RoboDK station: kr30 cnc_Test01.rdk

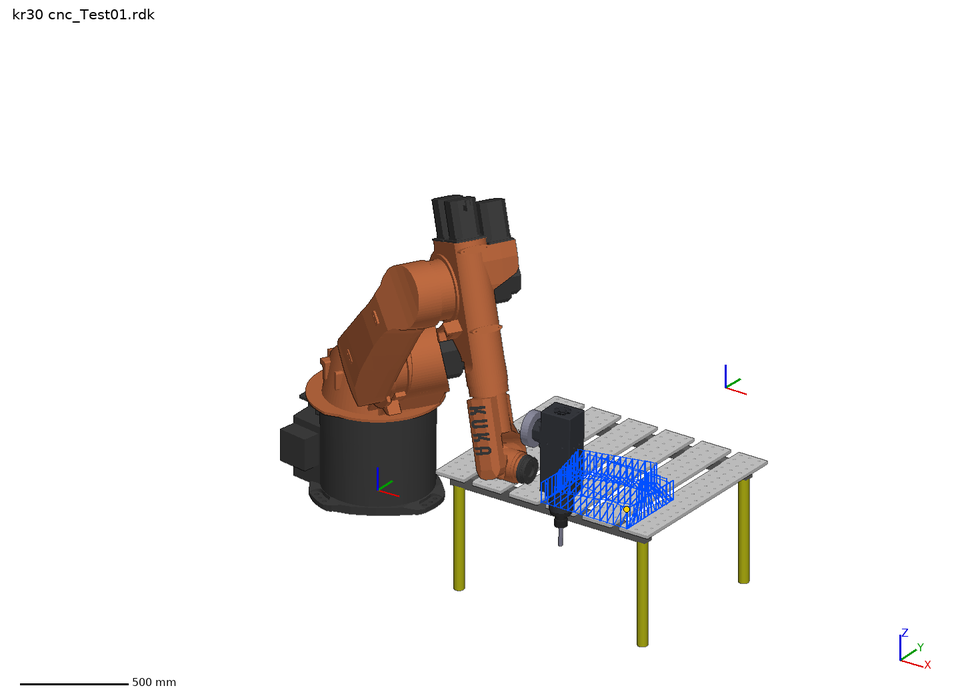
[picture v0: the station drawn from its stored meshes, robots at their saved joint values, targets as dots, program paths as lines]
Station kr30 cnc_Test01. Poses are relative to the parent item; angles as X-Y-Z fixed-axis rotations.
  - frame KUKA KR 30 HA Base at (0, 0, 0) mm
    - robot KUKA KR 30 HA: 6 axes, payload 30 kg, reach 2033 mm, repeatability 0.05 mm, weight 665 kg
        modified DH rows (alpha deg, a mm, theta deg, d mm): 0, 0, 0, 815; -90, 350, 0, 0; 0, 850, -90, 0; -90, 145, 0, 820; 90, 0, 0, 0; -90, 0, 180, 170
        joint limits [-185, -135, -120, -350, -119, -350] to [185, 35, 158, 350, 119, 350]; home [0, -90, 90, 0, 0, 0]; saved at [30.345, -48.669, 117.571, 35.552, -71.774, -11.781]
      - tool 1/2" End Mill TCP, TCP at (337.71, -2.2, 160.57) mm, size 692.9 x 170 x 256 mm
  - frame Milling Reference at (1256.02, 1000, 476.5) mm
    - object TABLE HEIGHT NOT YET SET at (0, -1000, 0) mm, size 1193.8 x 965.2 x 609.6 mm, geometry from welding_table.sld
    - object RhinoPart at (0, 0, 0) mm
  - machining project Machining Settings: rotZ(0) | rotX(0)*rotY(0) | rotZ(0) | onStart | onPathStart | onApproach | onPoint | onRetract | onFinish | Extruder(%1) | default | default | OutOnMov(%1) | OutOffMov(%1) | onPathFinish | M_RunCode(%1)
  - machining project RhinoPart Settings: rotZ(0) | rotX(0)*rotY(0) | roty(-90) | onStart | onPathStart | onApproach | onPoint | onRetract | onFinish | SetRPM(%1) | SetTool(%1) | Extruder(%1) | default | default | OutOnMov(%1) | OutOffMov(%1) | onPathFinish | M_RunCode(%1)
  - program RhinoPart (604 instructions, listed below)
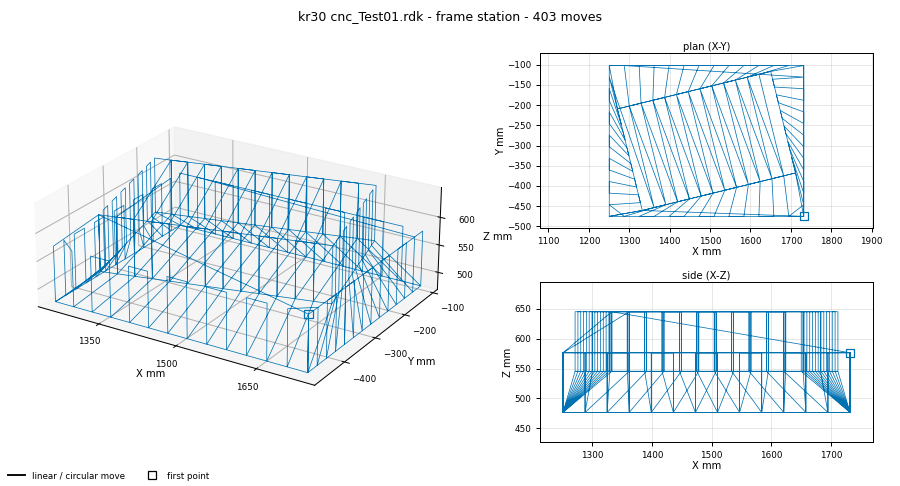
[picture p0: tool path of kr30 cnc_Test01.rdk in frame station, 403 of 403 moves have a stored position in this frame; points joined in program order, loops and branches not executed]

--- program RhinoPart (robot KUKA KR 30 HA) ---
  Set Ref.: Milling Reference
  Set Tool: 1/2" End Mill TCP
  Show 1/2" End Mill TCP
  Set speed (1000.0 mm/s)
  MoveJ 1 to (476.06, -1475.28, 100) mm, rotated rx 0 ry 90 rz 0 deg; joints [18.652, -58.205, 103.326, -154.528, 48.045, 162.335]
  MoveL 2 to (476.06, -1475.28, 100) mm, rotated rx 0 ry 90 rz 0 deg; joints [18.652, -58.205, 103.326, -154.528, 48.045, 162.335]
  MoveL 3 to (476.06, -1475.28, 0) mm, rotated rx 0 ry 90 rz 0 deg; joints [18.652, -54.047, 104.898, -156.478, 53.26, 165.406]
  MoveL 4 to (476.06, -1475.28, 0) mm, rotated rx 0 ry 90 rz 0 deg; joints [18.652, -54.047, 104.898, -156.478, 53.26, 165.406]
  Set speed (50.0 mm/s)
  MoveL 5 to (-5.57, -1475.28, 0) mm, rotated rx 0 ry 90 rz 0 deg; joints [27.216, -76.021, 140.928, -150.408, 67.844, 167.912]
  MoveL 6 to (-5.57, -1101.79, 0) mm, rotated rx 0 ry 90 rz 0 deg; joints [6.179, -81.84, 148.78, -173.289, 67.082, 177.377]
  MoveL 7 to (476.06, -1101.79, 0) mm, rotated rx 0 ry 90 rz 0 deg; joints [4.064, -57.785, 111.525, -174.964, 53.845, 177.024]
  MoveL 8 to (476.06, -1475.28, 0) mm, rotated rx 0 ry 90 rz 0 deg; joints [18.652, -54.047, 104.898, -156.478, 53.26, 165.406]
  Set speed (1000.0 mm/s)
  MoveL 9 to (476.06, -1475.28, 0) mm, rotated rx 0 ry 90 rz 0 deg; joints [18.652, -54.047, 104.898, -156.478, 53.26, 165.406]
  MoveL 10 to (476.06, -1475.28, 100) mm, rotated rx 0 ry 90 rz 0 deg; joints [18.652, -58.205, 103.326, -154.528, 48.045, 162.335]
  Set speed (1000.0 mm/s)
  MoveL 11 to (76.29, -1460.64, 168.91) mm, rotated rx 0 ry 90 rz 0 deg; joints [24.591, -82.592, 132.174, -148.989, 53.875, 160.486]
  MoveL 12 to (76.29, -1460.64, 68.91) mm, rotated rx 0 ry 90 rz 0 deg; joints [24.591, -77.019, 134.721, -151.568, 60.931, 165.262]
  MoveL 13 to (76.29, -1460.64, 68.91) mm, rotated rx 0 ry 90 rz 0 deg; joints [24.591, -77.019, 134.721, -151.568, 60.931, 165.262]
  Set speed (50.0 mm/s)
  MoveL 14 to (14.78, -1209.28, 68.91) mm, rotated rx 0 ry 90 rz 0 deg; joints [12.421, -85.064, 144.7, -165.681, 60.418, 172.818]
  MoveL 15 to (394.21, -1116.43, 68.91) mm, rotated rx 0 ry 90 rz 0 deg; joints [4.947, -65.156, 117.325, -173.745, 52.334, 176.169]
  MoveL 16 to (455.72, -1367.79, 68.91) mm, rotated rx 0 ry 90 rz 0 deg; joints [14.826, -59.674, 108.439, -160.608, 50.416, 167.358]
  MoveL 17 to (76.29, -1460.64, 68.91) mm, rotated rx 0 ry 90 rz 0 deg; joints [24.591, -77.019, 134.721, -151.568, 60.931, 165.262]
  Set speed (1000.0 mm/s)
  MoveL 18 to (76.29, -1460.64, 68.91) mm, rotated rx 0 ry 90 rz 0 deg; joints [24.591, -77.019, 134.721, -151.568, 60.931, 165.262]
  MoveL 19 to (76.29, -1460.64, 168.91) mm, rotated rx 0 ry 90 rz 0 deg; joints [24.591, -82.592, 132.174, -148.989, 53.875, 160.486]
  Set speed (1000.0 mm/s)
  MoveL 20 to (-5.57, -1475.28, 100) mm, rotated rx 0 ry 90 rz 0 deg; joints [27.216, -82.8, 138.885, -148.212, 60.252, 162.907]
  MoveL 21 to (-5.57, -1475.28, 0) mm, rotated rx 0 ry 90 rz 0 deg; joints [27.216, -76.021, 140.928, -150.408, 67.844, 167.912]
  MoveL 22 to (-5.57, -1475.28, 0) mm, rotated rx 0 ry 90 rz 0 deg; joints [27.216, -76.021, 140.928, -150.408, 67.844, 167.912]
  Set speed (50.0 mm/s)
  MoveL 23 to (76.29, -1460.64, 68.91) mm, rotated rx 0 ry 90 rz 0 deg; joints [24.591, -77.019, 134.721, -151.568, 60.931, 165.262]
  Set speed (1000.0 mm/s)
  MoveL 24 to (76.29, -1460.64, 68.91) mm, rotated rx 0 ry 90 rz 0 deg; joints [24.591, -77.019, 134.721, -151.568, 60.931, 165.262]
  MoveL 25 to (76.29, -1460.64, 168.91) mm, rotated rx 0 ry 90 rz 0 deg; joints [24.591, -82.592, 132.174, -148.989, 53.875, 160.486]
  Set speed (1000.0 mm/s)
  MoveL 26 to (455.72, -1367.79, 168.91) mm, rotated rx 0 ry 90 rz 0 deg; joints [14.826, -63.639, 106.295, -158.662, 44.688, 164.478]
  MoveL 27 to (455.72, -1367.79, 68.91) mm, rotated rx 0 ry 90 rz 0 deg; joints [14.826, -59.674, 108.439, -160.608, 50.416, 167.358]
  MoveL 28 to (455.72, -1367.79, 68.91) mm, rotated rx 0 ry 90 rz 0 deg; joints [14.826, -59.674, 108.439, -160.608, 50.416, 167.358]
  Set speed (50.0 mm/s)
  MoveL 29 to (476.06, -1475.28, 0) mm, rotated rx 0 ry 90 rz 0 deg; joints [18.652, -54.047, 104.898, -156.478, 53.26, 165.406]
  Set speed (1000.0 mm/s)
  MoveL 30 to (476.06, -1475.28, 0) mm, rotated rx 0 ry 90 rz 0 deg; joints [18.652, -54.047, 104.898, -156.478, 53.26, 165.406]
  MoveL 31 to (476.06, -1475.28, 100) mm, rotated rx 0 ry 90 rz 0 deg; joints [18.652, -58.205, 103.326, -154.528, 48.045, 162.335]
  Set speed (1000.0 mm/s)
  MoveL 32 to (476.06, -1101.79, 100) mm, rotated rx 0 ry 90 rz 0 deg; joints [4.064, -62.258, 109.929, -174.51, 47.803, 176.306]
  MoveL 33 to (476.06, -1101.79, 0) mm, rotated rx 0 ry 90 rz 0 deg; joints [4.064, -57.785, 111.525, -174.964, 53.845, 177.024]
  MoveL 34 to (476.06, -1101.79, 0) mm, rotated rx 0 ry 90 rz 0 deg; joints [4.064, -57.785, 111.525, -174.964, 53.845, 177.024]
  Set speed (50.0 mm/s)
  MoveL 35 to (394.21, -1116.43, 68.91) mm, rotated rx 0 ry 90 rz 0 deg; joints [4.947, -65.156, 117.325, -173.745, 52.334, 176.169]
  Set speed (1000.0 mm/s)
  MoveL 36 to (394.21, -1116.43, 68.91) mm, rotated rx 0 ry 90 rz 0 deg; joints [4.947, -65.156, 117.325, -173.745, 52.334, 176.169]
  MoveL 37 to (394.21, -1116.43, 168.91) mm, rotated rx 0 ry 90 rz 0 deg; joints [4.947, -69.559, 115.111, -173.086, 45.761, 175.165]
  Set speed (1000.0 mm/s)
  MoveL 38 to (14.78, -1209.28, 168.91) mm, rotated rx 0 ry 90 rz 0 deg; joints [12.421, -91.594, 141.782, -164.002, 51.297, 169.836]
  MoveL 39 to (14.78, -1209.28, 68.91) mm, rotated rx 0 ry 90 rz 0 deg; joints [12.421, -85.064, 144.7, -165.681, 60.418, 172.818]
  MoveL 40 to (14.78, -1209.28, 68.91) mm, rotated rx 0 ry 90 rz 0 deg; joints [12.421, -85.064, 144.7, -165.681, 60.418, 172.818]
  Set speed (50.0 mm/s)
  MoveL 41 to (-5.57, -1101.79, 0) mm, rotated rx 0 ry 90 rz 0 deg; joints [6.179, -81.84, 148.78, -173.289, 67.082, 177.377]
  Set speed (1000.0 mm/s)
  MoveL 42 to (-5.57, -1101.79, 0) mm, rotated rx 0 ry 90 rz 0 deg; joints [6.179, -81.84, 148.78, -173.289, 67.082, 177.377]
  MoveL 43 to (-5.57, -1101.79, 100) mm, rotated rx 0 ry 90 rz 0 deg; joints [6.179, -89.702, 146.455, -172.624, 56.97, 175.964]
  Set speed (1000.0 mm/s)
  MoveL 44 to (439.01, -1101.79, 100) mm, rotated rx 0 ry 90 rz 0 deg; joints [4.174, -64.255, 113.094, -174.463, 48.972, 176.359]
  MoveL 45 to (439.01, -1101.79, 0) mm, rotated rx 0 ry 90 rz 0 deg; joints [4.174, -59.613, 114.709, -174.914, 55.202, 177.093]
  MoveL 46 to (439.01, -1101.79, 0) mm, rotated rx 0 ry 90 rz 0 deg; joints [4.174, -59.613, 114.709, -174.914, 55.202, 177.093]
  Set speed (50.0 mm/s)
  MoveL 47 to (365.02, -1123.57, 68.91) mm, rotated rx 0 ry 90 rz 0 deg; joints [5.373, -66.644, 119.654, -173.284, 53.2, 175.965]
  Set speed (1000.0 mm/s)
  MoveL 48 to (365.02, -1123.57, 68.91) mm, rotated rx 0 ry 90 rz 0 deg; joints [5.373, -66.644, 119.654, -173.284, 53.2, 175.965]
  MoveL 49 to (365.02, -1123.57, 168.91) mm, rotated rx 0 ry 90 rz 0 deg; joints [5.373, -71.176, 117.413, -172.58, 46.477, 174.875]
  Set speed (1000.0 mm/s)
  MoveL 50 to (335.84, -1130.72, 168.91) mm, rotated rx 0 ry 90 rz 0 deg; joints [5.818, -72.795, 119.668, -172.052, 47.149, 174.576]
  MoveL 51 to (335.84, -1130.72, 68.91) mm, rotated rx 0 ry 90 rz 0 deg; joints [5.818, -68.13, 121.942, -172.805, 54.028, 175.759]
  MoveL 52 to (335.84, -1130.72, 68.91) mm, rotated rx 0 ry 90 rz 0 deg; joints [5.818, -68.13, 121.942, -172.805, 54.028, 175.759]
  Set speed (50.0 mm/s)
  MoveL 53 to (401.97, -1101.79, 0) mm, rotated rx 0 ry 90 rz 0 deg; joints [4.29, -61.424, 117.823, -174.853, 56.506, 177.154]
  Set speed (1000.0 mm/s)
  MoveL 54 to (401.97, -1101.79, 0) mm, rotated rx 0 ry 90 rz 0 deg; joints [4.29, -61.424, 117.823, -174.853, 56.506, 177.154]
  MoveL 55 to (401.97, -1101.79, 100) mm, rotated rx 0 ry 90 rz 0 deg; joints [4.29, -66.245, 116.184, -174.402, 50.074, 176.4]
  Set speed (1000.0 mm/s)
  MoveL 56 to (364.92, -1101.79, 100) mm, rotated rx 0 ry 90 rz 0 deg; joints [4.413, -68.234, 119.205, -174.326, 51.109, 176.431]
  MoveL 57 to (364.92, -1101.79, 0) mm, rotated rx 0 ry 90 rz 0 deg; joints [4.413, -63.224, 120.874, -174.78, 57.758, 177.21]
  MoveL 58 to (364.92, -1101.79, 0) mm, rotated rx 0 ry 90 rz 0 deg; joints [4.413, -63.224, 120.874, -174.78, 57.758, 177.21]
  Set speed (50.0 mm/s)
  MoveL 59 to (306.65, -1137.86, 68.91) mm, rotated rx 0 ry 90 rz 0 deg; joints [6.283, -69.615, 124.19, -172.305, 54.819, 175.548]
  Set speed (1000.0 mm/s)
  MoveL 60 to (306.65, -1137.86, 68.91) mm, rotated rx 0 ry 90 rz 0 deg; joints [6.283, -69.615, 124.19, -172.305, 54.819, 175.548]
  MoveL 61 to (306.65, -1137.86, 168.91) mm, rotated rx 0 ry 90 rz 0 deg; joints [6.283, -74.42, 121.88, -171.501, 47.775, 174.265]
  Set speed (1000.0 mm/s)
  MoveL 62 to (277.46, -1145, 168.91) mm, rotated rx 0 ry 90 rz 0 deg; joints [6.77, -76.052, 124.049, -170.924, 48.355, 173.94]
  MoveL 63 to (277.46, -1145, 68.91) mm, rotated rx 0 ry 90 rz 0 deg; joints [6.77, -71.103, 126.399, -171.783, 55.572, 175.333]
  MoveL 64 to (277.46, -1145, 68.91) mm, rotated rx 0 ry 90 rz 0 deg; joints [6.77, -71.103, 126.399, -171.783, 55.572, 175.333]
  Set speed (50.0 mm/s)
  MoveL 65 to (327.87, -1101.79, 0) mm, rotated rx 0 ry 90 rz 0 deg; joints [4.543, -65.017, 123.867, -174.696, 58.958, 177.259]
  Set speed (1000.0 mm/s)
  MoveL 66 to (327.87, -1101.79, 0) mm, rotated rx 0 ry 90 rz 0 deg; joints [4.543, -65.017, 123.867, -174.696, 58.958, 177.259]
  MoveL 67 to (327.87, -1101.79, 100) mm, rotated rx 0 ry 90 rz 0 deg; joints [4.543, -70.229, 122.163, -174.237, 52.075, 176.45]
  Set speed (1000.0 mm/s)
  MoveL 68 to (290.82, -1101.79, 100) mm, rotated rx 0 ry 90 rz 0 deg; joints [4.681, -72.237, 125.063, -174.133, 52.971, 176.459]
  MoveL 69 to (290.82, -1101.79, 0) mm, rotated rx 0 ry 90 rz 0 deg; joints [4.681, -66.809, 126.806, -174.599, 60.107, 177.302]
  MoveL 70 to (290.82, -1101.79, 0) mm, rotated rx 0 ry 90 rz 0 deg; joints [4.681, -66.809, 126.806, -174.599, 60.107, 177.302]
  Set speed (50.0 mm/s)
  MoveL 71 to (248.28, -1152.14, 68.91) mm, rotated rx 0 ry 90 rz 0 deg; joints [7.28, -72.596, 128.57, -171.237, 56.285, 175.11]
  Set speed (1000.0 mm/s)
  MoveL 72 to (248.28, -1152.14, 68.91) mm, rotated rx 0 ry 90 rz 0 deg; joints [7.28, -72.596, 128.57, -171.237, 56.285, 175.11]
  MoveL 73 to (248.28, -1152.14, 168.91) mm, rotated rx 0 ry 90 rz 0 deg; joints [7.28, -77.695, 126.177, -170.317, 48.889, 173.599]
  Set speed (1000.0 mm/s)
  MoveL 74 to (219.09, -1159.28, 168.91) mm, rotated rx 0 ry 90 rz 0 deg; joints [7.815, -79.352, 128.264, -169.68, 49.375, 173.238]
  MoveL 75 to (219.09, -1159.28, 68.91) mm, rotated rx 0 ry 90 rz 0 deg; joints [7.815, -74.097, 130.706, -170.665, 56.959, 174.878]
  MoveL 76 to (219.09, -1159.28, 68.91) mm, rotated rx 0 ry 90 rz 0 deg; joints [7.815, -74.097, 130.706, -170.665, 56.959, 174.878]
  Set speed (50.0 mm/s)
  MoveL 77 to (253.77, -1101.79, 0) mm, rotated rx 0 ry 90 rz 0 deg; joints [4.827, -68.606, 129.696, -174.489, 61.202, 177.339]
  Set speed (1000.0 mm/s)
  MoveL 78 to (253.77, -1101.79, 0) mm, rotated rx 0 ry 90 rz 0 deg; joints [4.827, -68.606, 129.696, -174.489, 61.202, 177.339]
  MoveL 79 to (253.77, -1101.79, 100) mm, rotated rx 0 ry 90 rz 0 deg; joints [4.827, -74.263, 127.907, -174.014, 53.793, 176.455]
  Set speed (1000.0 mm/s)
  MoveL 80 to (216.72, -1101.79, 100) mm, rotated rx 0 ry 90 rz 0 deg; joints [4.983, -76.315, 130.699, -173.878, 54.538, 176.439]
  MoveL 81 to (216.72, -1101.79, 0) mm, rotated rx 0 ry 90 rz 0 deg; joints [4.983, -70.411, 132.54, -174.367, 62.243, 177.37]
  MoveL 82 to (216.72, -1101.79, 0) mm, rotated rx 0 ry 90 rz 0 deg; joints [4.983, -70.411, 132.54, -174.367, 62.243, 177.37]
  Set speed (50.0 mm/s)
  MoveL 83 to (189.9, -1166.42, 68.91) mm, rotated rx 0 ry 90 rz 0 deg; joints [8.376, -75.608, 132.806, -170.064, 57.591, 174.637]
  Set speed (1000.0 mm/s)
  MoveL 84 to (189.9, -1166.42, 68.91) mm, rotated rx 0 ry 90 rz 0 deg; joints [8.376, -75.608, 132.806, -170.064, 57.591, 174.637]
  MoveL 85 to (189.9, -1166.42, 168.91) mm, rotated rx 0 ry 90 rz 0 deg; joints [8.376, -81.025, 130.312, -169.007, 49.811, 172.855]
  Set speed (1000.0 mm/s)
  MoveL 86 to (160.71, -1173.57, 168.91) mm, rotated rx 0 ry 90 rz 0 deg; joints [8.966, -82.718, 132.321, -168.296, 50.196, 172.445]
  MoveL 87 to (160.71, -1173.57, 68.91) mm, rotated rx 0 ry 90 rz 0 deg; joints [8.966, -77.132, 134.873, -169.432, 58.181, 174.382]
  MoveL 88 to (160.71, -1173.57, 68.91) mm, rotated rx 0 ry 90 rz 0 deg; joints [8.966, -77.132, 134.873, -169.432, 58.181, 174.382]
  Set speed (50.0 mm/s)
  MoveL 89 to (179.68, -1101.79, 0) mm, rotated rx 0 ry 90 rz 0 deg; joints [5.149, -72.232, 135.341, -174.23, 63.226, 177.394]
  Set speed (1000.0 mm/s)
  MoveL 90 to (179.68, -1101.79, 0) mm, rotated rx 0 ry 90 rz 0 deg; joints [5.149, -72.232, 135.341, -174.23, 63.226, 177.394]
  MoveL 91 to (179.68, -1101.79, 100) mm, rotated rx 0 ry 90 rz 0 deg; joints [5.149, -78.402, 133.441, -173.725, 55.2, 176.409]
  Set speed (1000.0 mm/s)
  MoveL 92 to (142.63, -1101.79, 100) mm, rotated rx 0 ry 90 rz 0 deg; joints [5.327, -80.532, 136.135, -173.553, 55.773, 176.363]
  MoveL 93 to (142.63, -1101.79, 0) mm, rotated rx 0 ry 90 rz 0 deg; joints [5.327, -74.075, 138.101, -174.079, 64.146, 177.41]
  MoveL 94 to (142.63, -1101.79, 0) mm, rotated rx 0 ry 90 rz 0 deg; joints [5.327, -74.075, 138.101, -174.079, 64.146, 177.41]
  Set speed (50.0 mm/s)
  MoveL 95 to (131.53, -1180.71, 68.91) mm, rotated rx 0 ry 90 rz 0 deg; joints [9.586, -78.673, 136.905, -168.765, 58.727, 174.112]
  Set speed (1000.0 mm/s)
  MoveL 96 to (131.53, -1180.71, 68.91) mm, rotated rx 0 ry 90 rz 0 deg; joints [9.586, -78.673, 136.905, -168.765, 58.727, 174.112]
  MoveL 97 to (131.53, -1180.71, 168.91) mm, rotated rx 0 ry 90 rz 0 deg; joints [9.586, -84.433, 134.291, -167.542, 50.529, 172.006]
  Set speed (1000.0 mm/s)
  MoveL 98 to (102.34, -1187.85, 168.91) mm, rotated rx 0 ry 90 rz 0 deg; joints [10.239, -86.175, 136.223, -166.741, 50.808, 171.531]
  MoveL 99 to (102.34, -1187.85, 68.91) mm, rotated rx 0 ry 90 rz 0 deg; joints [10.239, -80.232, 138.904, -168.06, 59.225, 173.825]
  MoveL 100 to (102.34, -1187.85, 68.91) mm, rotated rx 0 ry 90 rz 0 deg; joints [10.239, -80.232, 138.904, -168.06, 59.225, 173.825]
  Set speed (50.0 mm/s)
  MoveL 101 to (105.58, -1101.79, 0) mm, rotated rx 0 ry 90 rz 0 deg; joints [5.517, -75.948, 140.824, -173.91, 65, 177.418]
  Set speed (1000.0 mm/s)
  MoveL 102 to (105.58, -1101.79, 0) mm, rotated rx 0 ry 90 rz 0 deg; joints [5.517, -75.948, 140.824, -173.91, 65, 177.418]
  MoveL 103 to (105.58, -1101.79, 100) mm, rotated rx 0 ry 90 rz 0 deg; joints [5.517, -82.714, 138.783, -173.36, 56.248, 176.299]
  Set speed (1000.0 mm/s)
  MoveL 104 to (68.53, -1101.79, 100) mm, rotated rx 0 ry 90 rz 0 deg; joints [5.721, -84.961, 141.386, -173.143, 56.614, 176.214]
  MoveL 105 to (68.53, -1101.79, 0) mm, rotated rx 0 ry 90 rz 0 deg; joints [5.721, -77.859, 143.51, -173.724, 65.78, 177.417]
  MoveL 106 to (68.53, -1101.79, 0) mm, rotated rx 0 ry 90 rz 0 deg; joints [5.721, -77.859, 143.51, -173.724, 65.78, 177.417]
  Set speed (50.0 mm/s)
  MoveL 107 to (73.15, -1194.99, 68.91) mm, rotated rx 0 ry 90 rz 0 deg; joints [10.927, -81.815, 140.87, -167.314, 59.675, 173.516]
  Set speed (1000.0 mm/s)
  MoveL 108 to (73.15, -1194.99, 68.91) mm, rotated rx 0 ry 90 rz 0 deg; joints [10.927, -81.815, 140.87, -167.314, 59.675, 173.516]
  MoveL 109 to (73.15, -1194.99, 168.91) mm, rotated rx 0 ry 90 rz 0 deg; joints [10.927, -87.947, 138.116, -165.888, 51.03, 171.015]
  Set speed (1000.0 mm/s)
  MoveL 110 to (43.97, -1202.13, 168.91) mm, rotated rx 0 ry 90 rz 0 deg; joints [11.653, -89.752, 139.969, -164.977, 51.194, 170.453]
  MoveL 111 to (43.97, -1202.13, 68.91) mm, rotated rx 0 ry 90 rz 0 deg; joints [11.653, -83.424, 142.801, -166.522, 60.074, 173.182]
  MoveL 112 to (43.97, -1202.13, 68.91) mm, rotated rx 0 ry 90 rz 0 deg; joints [11.653, -83.424, 142.801, -166.522, 60.074, 173.182]
  Set speed (50.0 mm/s)
  MoveL 113 to (31.48, -1101.79, 0) mm, rotated rx 0 ry 90 rz 0 deg; joints [5.941, -79.819, 146.162, -173.518, 66.477, 177.404]
  Set speed (1000.0 mm/s)
  MoveL 114 to (31.48, -1101.79, 0) mm, rotated rx 0 ry 90 rz 0 deg; joints [5.941, -79.819, 146.162, -173.518, 66.477, 177.404]
  MoveL 115 to (31.48, -1101.79, 100) mm, rotated rx 0 ry 90 rz 0 deg; joints [5.941, -87.285, 143.943, -172.899, 56.86, 176.104]
  Set speed (1000.0 mm/s)
  MoveL 116 to (476.06, -1130.52, 100) mm, rotated rx 0 ry 90 rz 0 deg; joints [5.231, -62.132, 109.727, -172.932, 47.813, 175.24]
  MoveL 117 to (476.06, -1130.52, 0) mm, rotated rx 0 ry 90 rz 0 deg; joints [5.231, -57.67, 111.322, -173.515, 53.828, 176.162]
  MoveL 118 to (476.06, -1130.52, 0) mm, rotated rx 0 ry 90 rz 0 deg; joints [5.231, -57.67, 111.322, -173.515, 53.828, 176.162]
  Set speed (50.0 mm/s)
  MoveL 119 to (398.94, -1135.77, 68.91) mm, rotated rx 0 ry 90 rz 0 deg; joints [5.759, -64.815, 116.785, -172.704, 52.196, 175.513]
  Set speed (1000.0 mm/s)
  MoveL 120 to (398.94, -1135.77, 68.91) mm, rotated rx 0 ry 90 rz 0 deg; joints [5.759, -64.815, 116.785, -172.704, 52.196, 175.513]
  MoveL 121 to (398.94, -1135.77, 168.91) mm, rotated rx 0 ry 90 rz 0 deg; joints [5.759, -69.188, 114.577, -171.937, 45.673, 174.347]
  Set speed (1000.0 mm/s)
  MoveL 122 to (403.67, -1155.1, 168.91) mm, rotated rx 0 ry 90 rz 0 deg; joints [6.563, -68.804, 114.02, -170.793, 45.588, 173.529]
  MoveL 123 to (403.67, -1155.1, 68.91) mm, rotated rx 0 ry 90 rz 0 deg; joints [6.563, -64.46, 116.222, -171.667, 52.057, 174.854]
  MoveL 124 to (403.67, -1155.1, 68.91) mm, rotated rx 0 ry 90 rz 0 deg; joints [6.563, -64.46, 116.222, -171.667, 52.057, 174.854]
  Set speed (50.0 mm/s)
  MoveL 125 to (476.06, -1159.25, 0) mm, rotated rx 0 ry 90 rz 0 deg; joints [6.394, -57.525, 111.068, -172.069, 53.806, 175.297]
  Set speed (1000.0 mm/s)
  MoveL 126 to (476.06, -1159.25, 0) mm, rotated rx 0 ry 90 rz 0 deg; joints [6.394, -57.525, 111.068, -172.069, 53.806, 175.297]
  MoveL 127 to (476.06, -1159.25, 100) mm, rotated rx 0 ry 90 rz 0 deg; joints [6.394, -61.974, 109.474, -171.358, 47.826, 174.174]
  Set speed (1000.0 mm/s)
  MoveL 128 to (476.06, -1187.98, 100) mm, rotated rx 0 ry 90 rz 0 deg; joints [7.551, -61.785, 109.171, -169.789, 47.841, 173.107]
  MoveL 129 to (476.06, -1187.98, 0) mm, rotated rx 0 ry 90 rz 0 deg; joints [7.551, -57.351, 110.763, -170.626, 53.78, 174.428]
  MoveL 130 to (476.06, -1187.98, 0) mm, rotated rx 0 ry 90 rz 0 deg; joints [7.551, -57.351, 110.763, -170.626, 53.78, 174.428]
  Set speed (50.0 mm/s)
  MoveL 131 to (408.4, -1174.44, 68.91) mm, rotated rx 0 ry 90 rz 0 deg; joints [7.358, -64.091, 115.634, -170.636, 51.917, 174.192]
  Set speed (1000.0 mm/s)
  MoveL 132 to (408.4, -1174.44, 68.91) mm, rotated rx 0 ry 90 rz 0 deg; joints [7.358, -64.091, 115.634, -170.636, 51.917, 174.192]
  MoveL 133 to (408.4, -1174.44, 168.91) mm, rotated rx 0 ry 90 rz 0 deg; joints [7.358, -68.404, 113.438, -169.657, 45.504, 172.711]
  Set speed (1000.0 mm/s)
  MoveL 134 to (413.14, -1193.77, 168.91) mm, rotated rx 0 ry 90 rz 0 deg; joints [8.145, -67.99, 112.833, -168.527, 45.421, 171.893]
  MoveL 135 to (413.14, -1193.77, 68.91) mm, rotated rx 0 ry 90 rz 0 deg; joints [8.145, -63.709, 115.023, -169.61, 51.775, 173.528]
  MoveL 136 to (413.14, -1193.77, 68.91) mm, rotated rx 0 ry 90 rz 0 deg; joints [8.145, -63.709, 115.023, -169.61, 51.775, 173.528]
  Set speed (50.0 mm/s)
  MoveL 137 to (476.06, -1216.71, 0) mm, rotated rx 0 ry 90 rz 0 deg; joints [8.702, -57.148, 110.406, -169.187, 53.749, 173.556]
  Set speed (1000.0 mm/s)
  MoveL 138 to (476.06, -1216.71, 0) mm, rotated rx 0 ry 90 rz 0 deg; joints [8.702, -57.148, 110.406, -169.187, 53.749, 173.556]
  MoveL 139 to (476.06, -1216.71, 100) mm, rotated rx 0 ry 90 rz 0 deg; joints [8.702, -61.564, 108.816, -168.227, 47.858, 172.039]
  Set speed (1000.0 mm/s)
  MoveL 140 to (476.06, -1245.44, 100) mm, rotated rx 0 ry 90 rz 0 deg; joints [9.846, -61.313, 108.41, -166.671, 47.877, 170.97]
  MoveL 141 to (476.06, -1245.44, 0) mm, rotated rx 0 ry 90 rz 0 deg; joints [9.846, -56.917, 109.999, -167.752, 53.713, 172.679]
  MoveL 142 to (476.06, -1245.44, 0) mm, rotated rx 0 ry 90 rz 0 deg; joints [9.846, -56.917, 109.999, -167.752, 53.713, 172.679]
  Set speed (50.0 mm/s)
  MoveL 143 to (417.87, -1213.11, 68.91) mm, rotated rx 0 ry 90 rz 0 deg; joints [8.923, -63.313, 114.388, -168.59, 51.633, 172.86]
  Set speed (1000.0 mm/s)
  MoveL 144 to (417.87, -1213.11, 68.91) mm, rotated rx 0 ry 90 rz 0 deg; joints [8.923, -63.313, 114.388, -168.59, 51.633, 172.86]
  MoveL 145 to (417.87, -1213.11, 168.91) mm, rotated rx 0 ry 90 rz 0 deg; joints [8.923, -67.561, 112.203, -167.405, 45.34, 171.074]
  Set speed (1000.0 mm/s)
  MoveL 146 to (422.6, -1232.44, 168.91) mm, rotated rx 0 ry 90 rz 0 deg; joints [9.693, -67.119, 111.55, -166.289, 45.259, 170.255]
  MoveL 147 to (422.6, -1232.44, 68.91) mm, rotated rx 0 ry 90 rz 0 deg; joints [9.693, -62.904, 113.728, -167.575, 51.488, 172.188]
  MoveL 148 to (422.6, -1232.44, 68.91) mm, rotated rx 0 ry 90 rz 0 deg; joints [9.693, -62.904, 113.728, -167.575, 51.488, 172.188]
  Set speed (50.0 mm/s)
  MoveL 149 to (476.06, -1274.17, 0) mm, rotated rx 0 ry 90 rz 0 deg; joints [10.982, -56.657, 109.54, -166.322, 53.673, 171.797]
  Set speed (1000.0 mm/s)
  MoveL 150 to (476.06, -1274.17, 0) mm, rotated rx 0 ry 90 rz 0 deg; joints [10.982, -56.657, 109.54, -166.322, 53.673, 171.797]
  MoveL 151 to (476.06, -1274.17, 100) mm, rotated rx 0 ry 90 rz 0 deg; joints [10.982, -61.03, 107.954, -165.122, 47.897, 169.9]
  Set speed (1000.0 mm/s)
  MoveL 152 to (476.06, -1302.9, 100) mm, rotated rx 0 ry 90 rz 0 deg; joints [12.109, -60.717, 107.446, -163.581, 47.918, 168.829]
  MoveL 153 to (476.06, -1302.9, 0) mm, rotated rx 0 ry 90 rz 0 deg; joints [12.109, -56.368, 109.03, -164.898, 53.628, 170.908]
  MoveL 154 to (476.06, -1302.9, 0) mm, rotated rx 0 ry 90 rz 0 deg; joints [12.109, -56.368, 109.03, -164.898, 53.628, 170.908]
  Set speed (50.0 mm/s)
  MoveL 155 to (427.33, -1251.78, 68.91) mm, rotated rx 0 ry 90 rz 0 deg; joints [10.453, -62.481, 113.045, -166.565, 51.342, 171.513]
  Set speed (1000.0 mm/s)
  MoveL 156 to (427.33, -1251.78, 68.91) mm, rotated rx 0 ry 90 rz 0 deg; joints [10.453, -62.481, 113.045, -166.565, 51.342, 171.513]
  MoveL 157 to (427.33, -1251.78, 168.91) mm, rotated rx 0 ry 90 rz 0 deg; joints [10.453, -66.663, 110.872, -165.18, 45.178, 169.435]
  Set speed (1000.0 mm/s)
  MoveL 158 to (432.06, -1271.11, 168.91) mm, rotated rx 0 ry 90 rz 0 deg; joints [11.205, -66.192, 110.17, -164.077, 45.098, 168.614]
  MoveL 159 to (432.06, -1271.11, 68.91) mm, rotated rx 0 ry 90 rz 0 deg; joints [11.205, -62.045, 112.337, -165.56, 51.193, 170.833]
  MoveL 160 to (432.06, -1271.11, 68.91) mm, rotated rx 0 ry 90 rz 0 deg; joints [11.205, -62.045, 112.337, -165.56, 51.193, 170.833]
  Set speed (50.0 mm/s)
  MoveL 161 to (476.06, -1331.63, 0) mm, rotated rx 0 ry 90 rz 0 deg; joints [13.228, -56.052, 108.47, -163.479, 53.579, 170.013]
  Set speed (1000.0 mm/s)
  MoveL 162 to (476.06, -1331.63, 0) mm, rotated rx 0 ry 90 rz 0 deg; joints [13.228, -56.052, 108.47, -163.479, 53.579, 170.013]
  MoveL 163 to (476.06, -1331.63, 100) mm, rotated rx 0 ry 90 rz 0 deg; joints [13.228, -60.373, 106.888, -162.049, 47.939, 167.755]
  Set speed (1000.0 mm/s)
  MoveL 164 to (476.06, -1360.36, 100) mm, rotated rx 0 ry 90 rz 0 deg; joints [14.335, -59.999, 106.278, -160.526, 47.961, 166.679]
  MoveL 165 to (476.06, -1360.36, 0) mm, rotated rx 0 ry 90 rz 0 deg; joints [14.335, -55.707, 107.858, -162.067, 53.525, 169.11]
  MoveL 166 to (476.06, -1360.36, 0) mm, rotated rx 0 ry 90 rz 0 deg; joints [14.335, -55.707, 107.858, -162.067, 53.525, 169.11]
  Set speed (50.0 mm/s)
  MoveL 167 to (436.79, -1290.45, 68.91) mm, rotated rx 0 ry 90 rz 0 deg; joints [11.948, -61.597, 111.606, -164.56, 51.043, 170.149]
  Set speed (1000.0 mm/s)
  MoveL 168 to (436.79, -1290.45, 68.91) mm, rotated rx 0 ry 90 rz 0 deg; joints [11.948, -61.597, 111.606, -164.56, 51.043, 170.149]
  MoveL 169 to (436.79, -1290.45, 168.91) mm, rotated rx 0 ry 90 rz 0 deg; joints [11.948, -65.709, 109.444, -162.982, 45.018, 167.791]
  Set speed (1000.0 mm/s)
  MoveL 170 to (441.52, -1309.79, 168.91) mm, rotated rx 0 ry 90 rz 0 deg; joints [12.681, -65.211, 108.693, -161.893, 44.937, 166.967]
  MoveL 171 to (441.52, -1309.79, 68.91) mm, rotated rx 0 ry 90 rz 0 deg; joints [12.681, -61.135, 110.851, -163.566, 50.89, 169.459]
  MoveL 172 to (441.52, -1309.79, 68.91) mm, rotated rx 0 ry 90 rz 0 deg; joints [12.681, -61.135, 110.851, -163.566, 50.89, 169.459]
  Set speed (50.0 mm/s)
  MoveL 173 to (476.06, -1389.09, 0) mm, rotated rx 0 ry 90 rz 0 deg; joints [15.432, -55.334, 107.195, -160.66, 53.466, 168.198]
  Set speed (1000.0 mm/s)
  MoveL 174 to (476.06, -1389.09, 0) mm, rotated rx 0 ry 90 rz 0 deg; joints [15.432, -55.334, 107.195, -160.66, 53.466, 168.198]
  MoveL 175 to (476.06, -1389.09, 100) mm, rotated rx 0 ry 90 rz 0 deg; joints [15.432, -59.595, 105.617, -159.012, 47.983, 165.599]
  Set speed (1000.0 mm/s)
  MoveL 176 to (476.06, -1417.82, 100) mm, rotated rx 0 ry 90 rz 0 deg; joints [16.518, -59.161, 104.905, -157.508, 48.005, 164.516]
  MoveL 177 to (476.06, -1417.82, 0) mm, rotated rx 0 ry 90 rz 0 deg; joints [16.518, -54.933, 106.481, -159.259, 53.402, 167.278]
  MoveL 178 to (476.06, -1417.82, 0) mm, rotated rx 0 ry 90 rz 0 deg; joints [16.518, -54.933, 106.481, -159.259, 53.402, 167.278]
  Set speed (50.0 mm/s)
  MoveL 179 to (446.25, -1329.12, 68.91) mm, rotated rx 0 ry 90 rz 0 deg; joints [13.405, -60.661, 110.071, -162.575, 50.734, 168.765]
  Set speed (1000.0 mm/s)
  MoveL 180 to (446.25, -1329.12, 68.91) mm, rotated rx 0 ry 90 rz 0 deg; joints [13.405, -60.661, 110.071, -162.575, 50.734, 168.765]
  MoveL 181 to (446.25, -1329.12, 168.91) mm, rotated rx 0 ry 90 rz 0 deg; joints [13.405, -64.7, 107.919, -160.81, 44.855, 166.14]
  Set speed (1000.0 mm/s)
  MoveL 182 to (450.99, -1348.46, 168.91) mm, rotated rx 0 ry 90 rz 0 deg; joints [14.12, -64.176, 107.119, -159.733, 44.772, 165.311]
  MoveL 183 to (450.99, -1348.46, 68.91) mm, rotated rx 0 ry 90 rz 0 deg; joints [14.12, -60.174, 109.267, -161.59, 50.577, 168.065]
  MoveL 184 to (450.99, -1348.46, 68.91) mm, rotated rx 0 ry 90 rz 0 deg; joints [14.12, -60.174, 109.267, -161.59, 50.577, 168.065]
  Set speed (50.0 mm/s)
  MoveL 185 to (476.06, -1446.55, 0) mm, rotated rx 0 ry 90 rz 0 deg; joints [17.591, -54.504, 105.715, -157.865, 53.333, 166.347]
  Set speed (1000.0 mm/s)
  MoveL 186 to (476.06, -1446.55, 0) mm, rotated rx 0 ry 90 rz 0 deg; joints [17.591, -54.504, 105.715, -157.865, 53.333, 166.347]
  MoveL 187 to (476.06, -1446.55, 100) mm, rotated rx 0 ry 90 rz 0 deg; joints [17.591, -58.698, 104.141, -156.013, 48.025, 163.428]
  Set speed (1000.0 mm/s)
  MoveL 188 to (439.01, -1475.28, 100) mm, rotated rx 0 ry 90 rz 0 deg; joints [19.122, -60.131, 106.492, -154.402, 49.306, 162.653]
  MoveL 189 to (439.01, -1475.28, 0) mm, rotated rx 0 ry 90 rz 0 deg; joints [19.122, -55.828, 108.073, -156.321, 54.655, 165.765]
  MoveL 190 to (439.01, -1475.28, 0) mm, rotated rx 0 ry 90 rz 0 deg; joints [19.122, -55.828, 108.073, -156.321, 54.655, 165.765]
  Set speed (50.0 mm/s)
  MoveL 191 to (426.53, -1374.93, 68.91) mm, rotated rx 0 ry 90 rz 0 deg; joints [15.413, -61.068, 110.741, -160.118, 51.4, 167.286]
  Set speed (1000.0 mm/s)
  MoveL 192 to (426.53, -1374.93, 68.91) mm, rotated rx 0 ry 90 rz 0 deg; joints [15.413, -61.068, 110.741, -160.118, 51.4, 167.286]
  MoveL 193 to (426.53, -1374.93, 168.91) mm, rotated rx 0 ry 90 rz 0 deg; joints [15.413, -65.139, 108.584, -158.153, 45.579, 164.325]
  Set speed (1000.0 mm/s)
  MoveL 194 to (397.34, -1382.08, 168.91) mm, rotated rx 0 ry 90 rz 0 deg; joints [16.023, -66.626, 110.817, -157.609, 46.436, 164.149]
  MoveL 195 to (397.34, -1382.08, 68.91) mm, rotated rx 0 ry 90 rz 0 deg; joints [16.023, -62.447, 112.99, -159.597, 52.351, 167.2]
  MoveL 196 to (397.34, -1382.08, 68.91) mm, rotated rx 0 ry 90 rz 0 deg; joints [16.023, -62.447, 112.99, -159.597, 52.351, 167.2]
  Set speed (50.0 mm/s)
  MoveL 197 to (401.97, -1475.28, 0) mm, rotated rx 0 ry 90 rz 0 deg; joints [19.616, -57.579, 111.163, -156.113, 56, 166.09]
  Set speed (1000.0 mm/s)
  MoveL 198 to (401.97, -1475.28, 0) mm, rotated rx 0 ry 90 rz 0 deg; joints [19.616, -57.579, 111.163, -156.113, 56, 166.09]
  MoveL 199 to (401.97, -1475.28, 100) mm, rotated rx 0 ry 90 rz 0 deg; joints [19.616, -62.033, 109.569, -154.214, 50.51, 162.921]
  Set speed (1000.0 mm/s)
  MoveL 200 to (364.92, -1475.28, 100) mm, rotated rx 0 ry 90 rz 0 deg; joints [20.134, -63.917, 112.563, -153.968, 51.659, 163.144]
  MoveL 201 to (364.92, -1475.28, 0) mm, rotated rx 0 ry 90 rz 0 deg; joints [20.134, -59.304, 114.174, -155.854, 57.298, 166.385]
  MoveL 202 to (364.92, -1475.28, 0) mm, rotated rx 0 ry 90 rz 0 deg; joints [20.134, -59.304, 114.174, -155.854, 57.298, 166.385]
  Set speed (50.0 mm/s)
  MoveL 203 to (368.16, -1389.22, 68.91) mm, rotated rx 0 ry 90 rz 0 deg; joints [16.656, -63.812, 115.188, -159.046, 53.272, 167.101]
  Set speed (1000.0 mm/s)
  MoveL 204 to (368.16, -1389.22, 68.91) mm, rotated rx 0 ry 90 rz 0 deg; joints [16.656, -63.812, 115.188, -159.046, 53.272, 167.101]
  MoveL 205 to (368.16, -1389.22, 168.91) mm, rotated rx 0 ry 90 rz 0 deg; joints [16.656, -68.101, 112.996, -157.029, 47.259, 163.951]
  Set speed (1000.0 mm/s)
  MoveL 206 to (338.97, -1396.36, 168.91) mm, rotated rx 0 ry 90 rz 0 deg; joints [17.314, -69.568, 115.124, -156.412, 48.05, 163.728]
  MoveL 207 to (338.97, -1396.36, 68.91) mm, rotated rx 0 ry 90 rz 0 deg; joints [17.314, -65.165, 117.338, -158.463, 54.163, 166.989]
  MoveL 208 to (338.97, -1396.36, 68.91) mm, rotated rx 0 ry 90 rz 0 deg; joints [17.314, -65.165, 117.338, -158.463, 54.163, 166.989]
  Set speed (50.0 mm/s)
  MoveL 209 to (327.87, -1475.28, 0) mm, rotated rx 0 ry 90 rz 0 deg; joints [20.68, -61.009, 117.114, -155.546, 58.55, 166.653]
  Set speed (1000.0 mm/s)
  MoveL 210 to (327.87, -1475.28, 0) mm, rotated rx 0 ry 90 rz 0 deg; joints [20.68, -61.009, 117.114, -155.546, 58.55, 166.653]
  MoveL 211 to (327.87, -1475.28, 100) mm, rotated rx 0 ry 90 rz 0 deg; joints [20.68, -65.788, 115.48, -153.665, 52.756, 163.323]
  Set speed (1000.0 mm/s)
  MoveL 212 to (290.82, -1475.28, 100) mm, rotated rx 0 ry 90 rz 0 deg; joints [21.254, -67.65, 118.326, -153.306, 53.8, 163.46]
  MoveL 213 to (290.82, -1475.28, 0) mm, rotated rx 0 ry 90 rz 0 deg; joints [21.254, -62.697, 119.986, -155.19, 59.758, 166.894]
  MoveL 214 to (290.82, -1475.28, 0) mm, rotated rx 0 ry 90 rz 0 deg; joints [21.254, -62.697, 119.986, -155.19, 59.758, 166.894]
  Set speed (50.0 mm/s)
  MoveL 215 to (309.78, -1403.5, 68.91) mm, rotated rx 0 ry 90 rz 0 deg; joints [17.998, -66.507, 119.442, -157.846, 55.024, 166.863]
  Set speed (1000.0 mm/s)
  MoveL 216 to (309.78, -1403.5, 68.91) mm, rotated rx 0 ry 90 rz 0 deg; joints [17.998, -66.507, 119.442, -157.846, 55.024, 166.863]
  MoveL 217 to (309.78, -1403.5, 168.91) mm, rotated rx 0 ry 90 rz 0 deg; joints [17.998, -71.027, 117.202, -155.758, 48.809, 163.482]
  Set speed (1000.0 mm/s)
  MoveL 218 to (280.59, -1410.64, 168.91) mm, rotated rx 0 ry 90 rz 0 deg; joints [18.709, -72.48, 119.233, -155.064, 49.538, 163.21]
  MoveL 219 to (280.59, -1410.64, 68.91) mm, rotated rx 0 ry 90 rz 0 deg; joints [18.709, -67.841, 121.5, -157.196, 55.856, 166.722]
  MoveL 220 to (280.59, -1410.64, 68.91) mm, rotated rx 0 ry 90 rz 0 deg; joints [18.709, -67.841, 121.5, -157.196, 55.856, 166.722]
  Set speed (50.0 mm/s)
  MoveL 221 to (253.77, -1475.28, 0) mm, rotated rx 0 ry 90 rz 0 deg; joints [21.86, -64.371, 122.795, -154.784, 60.923, 167.11]
  Set speed (1000.0 mm/s)
  MoveL 222 to (253.77, -1475.28, 0) mm, rotated rx 0 ry 90 rz 0 deg; joints [21.86, -64.371, 122.795, -154.784, 60.923, 167.11]
  MoveL 223 to (253.77, -1475.28, 100) mm, rotated rx 0 ry 90 rz 0 deg; joints [21.86, -69.509, 121.104, -152.89, 54.792, 163.555]
  Set speed (1000.0 mm/s)
  MoveL 224 to (216.72, -1475.28, 100) mm, rotated rx 0 ry 90 rz 0 deg; joints [22.499, -71.369, 123.819, -152.416, 55.732, 163.608]
  MoveL 225 to (216.72, -1475.28, 0) mm, rotated rx 0 ry 90 rz 0 deg; joints [22.499, -66.036, 125.544, -154.328, 62.044, 167.301]
  MoveL 226 to (216.72, -1475.28, 0) mm, rotated rx 0 ry 90 rz 0 deg; joints [22.499, -66.036, 125.544, -154.328, 62.044, 167.301]
  Set speed (50.0 mm/s)
  MoveL 227 to (251.41, -1417.78, 68.91) mm, rotated rx 0 ry 90 rz 0 deg; joints [19.45, -69.166, 123.515, -156.511, 56.661, 166.567]
  Set speed (1000.0 mm/s)
  MoveL 228 to (251.41, -1417.78, 68.91) mm, rotated rx 0 ry 90 rz 0 deg; joints [19.45, -69.166, 123.515, -156.511, 56.661, 166.567]
  MoveL 229 to (251.41, -1417.78, 168.91) mm, rotated rx 0 ry 90 rz 0 deg; joints [19.45, -73.928, 121.216, -154.331, 50.237, 162.913]
  Set speed (1000.0 mm/s)
  MoveL 230 to (222.22, -1424.93, 168.91) mm, rotated rx 0 ry 90 rz 0 deg; joints [20.221, -75.374, 123.154, -153.556, 50.908, 162.587]
  MoveL 231 to (222.22, -1424.93, 68.91) mm, rotated rx 0 ry 90 rz 0 deg; joints [20.221, -70.485, 125.486, -155.789, 57.438, 166.396]
  MoveL 232 to (222.22, -1424.93, 68.91) mm, rotated rx 0 ry 90 rz 0 deg; joints [20.221, -70.485, 125.486, -155.789, 57.438, 166.396]
  Set speed (50.0 mm/s)
  MoveL 233 to (179.68, -1475.28, 0) mm, rotated rx 0 ry 90 rz 0 deg; joints [23.175, -67.695, 128.237, -153.819, 63.122, 167.469]
  Set speed (1000.0 mm/s)
  MoveL 234 to (179.68, -1475.28, 0) mm, rotated rx 0 ry 90 rz 0 deg; joints [23.175, -67.695, 128.237, -153.819, 63.122, 167.469]
  MoveL 235 to (179.68, -1475.28, 100) mm, rotated rx 0 ry 90 rz 0 deg; joints [23.175, -73.233, 126.472, -151.882, 56.62, 163.617]
  Set speed (1000.0 mm/s)
  MoveL 236 to (142.63, -1475.28, 100) mm, rotated rx 0 ry 90 rz 0 deg; joints [23.89, -75.108, 129.067, -151.287, 57.456, 163.581]
  MoveL 237 to (142.63, -1475.28, 0) mm, rotated rx 0 ry 90 rz 0 deg; joints [23.89, -69.35, 130.877, -153.257, 64.157, 167.612]
  MoveL 238 to (142.63, -1475.28, 0) mm, rotated rx 0 ry 90 rz 0 deg; joints [23.89, -69.35, 130.877, -153.257, 64.157, 167.612]
  Set speed (50.0 mm/s)
  MoveL 239 to (193.03, -1432.07, 68.91) mm, rotated rx 0 ry 90 rz 0 deg; joints [21.023, -71.799, 127.416, -155.029, 58.188, 166.208]
  Set speed (1000.0 mm/s)
  MoveL 240 to (193.03, -1432.07, 68.91) mm, rotated rx 0 ry 90 rz 0 deg; joints [21.023, -71.799, 127.416, -155.029, 58.188, 166.208]
  MoveL 241 to (193.03, -1432.07, 168.91) mm, rotated rx 0 ry 90 rz 0 deg; joints [21.023, -76.817, 125.046, -152.737, 51.552, 162.233]
  Set speed (1000.0 mm/s)
  MoveL 242 to (163.85, -1439.21, 168.91) mm, rotated rx 0 ry 90 rz 0 deg; joints [21.86, -78.26, 126.894, -151.873, 52.169, 161.848]
  MoveL 243 to (163.85, -1439.21, 68.91) mm, rotated rx 0 ry 90 rz 0 deg; joints [21.86, -73.108, 129.304, -154.228, 58.912, 166.001]
  MoveL 244 to (163.85, -1439.21, 68.91) mm, rotated rx 0 ry 90 rz 0 deg; joints [21.86, -73.108, 129.304, -154.228, 58.912, 166.001]
  Set speed (50.0 mm/s)
  MoveL 245 to (105.58, -1475.28, 0) mm, rotated rx 0 ry 90 rz 0 deg; joints [24.648, -71.007, 133.464, -152.638, 65.148, 167.73]
  Set speed (1000.0 mm/s)
  MoveL 246 to (105.58, -1475.28, 0) mm, rotated rx 0 ry 90 rz 0 deg; joints [24.648, -71.007, 133.464, -152.638, 65.148, 167.73]
  MoveL 247 to (105.58, -1475.28, 100) mm, rotated rx 0 ry 90 rz 0 deg; joints [24.648, -76.997, 131.605, -150.627, 58.238, 163.496]
  Set speed (1000.0 mm/s)
  MoveL 248 to (68.53, -1475.28, 100) mm, rotated rx 0 ry 90 rz 0 deg; joints [25.452, -78.905, 134.087, -149.897, 58.965, 163.359]
  MoveL 249 to (68.53, -1475.28, 0) mm, rotated rx 0 ry 90 rz 0 deg; joints [25.452, -72.669, 136.001, -151.96, 66.093, 167.82]
  MoveL 250 to (68.53, -1475.28, 0) mm, rotated rx 0 ry 90 rz 0 deg; joints [25.452, -72.669, 136.001, -151.96, 66.093, 167.82]
  Set speed (50.0 mm/s)
  MoveL 251 to (134.66, -1446.35, 68.91) mm, rotated rx 0 ry 90 rz 0 deg; joints [22.732, -74.414, 131.151, -153.386, 59.61, 165.776]
  Set speed (1000.0 mm/s)
  MoveL 252 to (134.66, -1446.35, 68.91) mm, rotated rx 0 ry 90 rz 0 deg; joints [22.732, -74.414, 131.151, -153.386, 59.61, 165.776]
  MoveL 253 to (134.66, -1446.35, 168.91) mm, rotated rx 0 ry 90 rz 0 deg; joints [22.732, -79.702, 128.698, -150.962, 52.76, 161.429]
  Set speed (1000.0 mm/s)
  MoveL 254 to (105.47, -1453.49, 168.91) mm, rotated rx 0 ry 90 rz 0 deg; joints [23.642, -81.146, 130.458, -150.001, 53.329, 160.976]
  MoveL 255 to (105.47, -1453.49, 68.91) mm, rotated rx 0 ry 90 rz 0 deg; joints [23.642, -75.717, 132.956, -152.5, 60.283, 165.53]
  MoveL 256 to (105.47, -1453.49, 68.91) mm, rotated rx 0 ry 90 rz 0 deg; joints [23.642, -75.717, 132.956, -152.5, 60.283, 165.53]
  Set speed (50.0 mm/s)
  MoveL 257 to (31.48, -1475.28, 0) mm, rotated rx 0 ry 90 rz 0 deg; joints [26.307, -74.339, 138.489, -151.218, 66.992, 167.882]
  Set speed (1000.0 mm/s)
  MoveL 258 to (31.48, -1475.28, 0) mm, rotated rx 0 ry 90 rz 0 deg; joints [26.307, -74.339, 138.489, -151.218, 66.992, 167.882]
  MoveL 259 to (31.48, -1475.28, 100) mm, rotated rx 0 ry 90 rz 0 deg; joints [26.307, -80.837, 136.513, -149.094, 59.637, 163.165]
  Set speed (1000.0 mm/s)
  MoveL 260 to (-5.57, -1446.55, 100) mm, rotated rx 0 ry 90 rz 0 deg; joints [25.783, -83.574, 139.794, -149.836, 59.957, 163.777]
  MoveL 261 to (-5.57, -1446.55, 0) mm, rotated rx 0 ry 90 rz 0 deg; joints [25.783, -76.681, 141.866, -151.978, 67.795, 168.628]
  MoveL 262 to (-5.57, -1446.55, 0) mm, rotated rx 0 ry 90 rz 0 deg; joints [25.783, -76.681, 141.866, -151.978, 67.795, 168.628]
  Set speed (50.0 mm/s)
  MoveL 263 to (71.55, -1441.3, 68.91) mm, rotated rx 0 ry 90 rz 0 deg; joints [23.77, -77.697, 135.624, -152.537, 60.925, 165.825]
  Set speed (1000.0 mm/s)
  MoveL 264 to (71.55, -1441.3, 68.91) mm, rotated rx 0 ry 90 rz 0 deg; joints [23.77, -77.697, 135.624, -152.537, 60.925, 165.825]
  MoveL 265 to (71.55, -1441.3, 168.91) mm, rotated rx 0 ry 90 rz 0 deg; joints [23.77, -83.346, 133.05, -149.996, 53.71, 161.131]
  Set speed (1000.0 mm/s)
  MoveL 266 to (66.82, -1421.96, 168.91) mm, rotated rx 0 ry 90 rz 0 deg; joints [22.93, -84.092, 133.904, -151.024, 53.537, 161.784]
  MoveL 267 to (66.82, -1421.96, 68.91) mm, rotated rx 0 ry 90 rz 0 deg; joints [22.93, -78.366, 136.506, -153.523, 60.912, 166.388]
  MoveL 268 to (66.82, -1421.96, 68.91) mm, rotated rx 0 ry 90 rz 0 deg; joints [22.93, -78.366, 136.506, -153.523, 60.912, 166.388]
  Set speed (50.0 mm/s)
  MoveL 269 to (-5.57, -1417.82, 0) mm, rotated rx 0 ry 90 rz 0 deg; joints [24.315, -77.312, 142.751, -153.583, 67.741, 169.343]
  Set speed (1000.0 mm/s)
  MoveL 270 to (-5.57, -1417.82, 0) mm, rotated rx 0 ry 90 rz 0 deg; joints [24.315, -77.312, 142.751, -153.583, 67.741, 169.343]
  MoveL 271 to (-5.57, -1417.82, 100) mm, rotated rx 0 ry 90 rz 0 deg; joints [24.315, -84.316, 140.652, -151.504, 59.658, 164.665]
  Set speed (1000.0 mm/s)
  MoveL 272 to (-5.57, -1389.09, 100) mm, rotated rx 0 ry 90 rz 0 deg; joints [22.811, -85.024, 141.458, -153.217, 59.358, 165.573]
  MoveL 273 to (-5.57, -1389.09, 0) mm, rotated rx 0 ry 90 rz 0 deg; joints [22.811, -77.913, 143.584, -155.223, 67.682, 170.058]
  MoveL 274 to (-5.57, -1389.09, 0) mm, rotated rx 0 ry 90 rz 0 deg; joints [22.811, -77.913, 143.584, -155.223, 67.682, 170.058]
  Set speed (50.0 mm/s)
  MoveL 275 to (62.09, -1402.63, 68.91) mm, rotated rx 0 ry 90 rz 0 deg; joints [22.072, -79.028, 137.365, -154.527, 60.893, 166.953]
  Set speed (1000.0 mm/s)
  MoveL 276 to (62.09, -1402.63, 68.91) mm, rotated rx 0 ry 90 rz 0 deg; joints [22.072, -79.028, 137.365, -154.527, 60.893, 166.953]
  MoveL 277 to (62.09, -1402.63, 168.91) mm, rotated rx 0 ry 90 rz 0 deg; joints [22.072, -84.829, 134.737, -152.074, 53.357, 162.445]
  Set speed (1000.0 mm/s)
  MoveL 278 to (57.36, -1383.29, 168.91) mm, rotated rx 0 ry 90 rz 0 deg; joints [21.194, -85.558, 135.546, -153.148, 53.169, 163.118]
  MoveL 279 to (57.36, -1383.29, 68.91) mm, rotated rx 0 ry 90 rz 0 deg; joints [21.194, -79.68, 138.203, -155.55, 60.867, 167.519]
  MoveL 280 to (57.36, -1383.29, 68.91) mm, rotated rx 0 ry 90 rz 0 deg; joints [21.194, -79.68, 138.203, -155.55, 60.867, 167.519]
  Set speed (50.0 mm/s)
  MoveL 281 to (-5.57, -1360.36, 0) mm, rotated rx 0 ry 90 rz 0 deg; joints [21.274, -78.481, 144.363, -156.897, 67.618, 170.774]
  Set speed (1000.0 mm/s)
  MoveL 282 to (-5.57, -1360.36, 0) mm, rotated rx 0 ry 90 rz 0 deg; joints [21.274, -78.481, 144.363, -156.897, 67.618, 170.774]
  MoveL 283 to (-5.57, -1360.36, 100) mm, rotated rx 0 ry 90 rz 0 deg; joints [21.274, -85.696, 142.21, -154.975, 59.06, 166.503]
  Set speed (1000.0 mm/s)
  MoveL 284 to (-5.57, -1331.63, 100) mm, rotated rx 0 ry 90 rz 0 deg; joints [19.704, -86.329, 142.908, -156.777, 58.766, 167.457]
  MoveL 285 to (-5.57, -1331.63, 0) mm, rotated rx 0 ry 90 rz 0 deg; joints [19.704, -79.015, 145.087, -158.605, 67.552, 171.491]
  MoveL 286 to (-5.57, -1331.63, 0) mm, rotated rx 0 ry 90 rz 0 deg; joints [19.704, -79.015, 145.087, -158.605, 67.552, 171.491]
  Set speed (50.0 mm/s)
  MoveL 287 to (52.63, -1363.96, 68.91) mm, rotated rx 0 ry 90 rz 0 deg; joints [20.298, -80.323, 139.018, -156.593, 60.835, 168.088]
  Set speed (1000.0 mm/s)
  MoveL 288 to (52.63, -1363.96, 68.91) mm, rotated rx 0 ry 90 rz 0 deg; joints [20.298, -80.323, 139.018, -156.593, 60.835, 168.088]
  MoveL 289 to (52.63, -1363.96, 168.91) mm, rotated rx 0 ry 90 rz 0 deg; joints [20.298, -86.277, 136.333, -154.246, 52.975, 163.801]
  Set speed (1000.0 mm/s)
  MoveL 290 to (47.9, -1344.62, 168.91) mm, rotated rx 0 ry 90 rz 0 deg; joints [19.382, -86.985, 137.097, -155.369, 52.775, 164.498]
  MoveL 291 to (47.9, -1344.62, 68.91) mm, rotated rx 0 ry 90 rz 0 deg; joints [19.382, -80.956, 139.811, -157.655, 60.798, 168.66]
  MoveL 292 to (47.9, -1344.62, 68.91) mm, rotated rx 0 ry 90 rz 0 deg; joints [19.382, -80.956, 139.811, -157.655, 60.798, 168.66]
  Set speed (50.0 mm/s)
  MoveL 293 to (-5.57, -1302.9, 0) mm, rotated rx 0 ry 90 rz 0 deg; joints [18.102, -79.513, 145.755, -160.345, 67.484, 172.212]
  Set speed (1000.0 mm/s)
  MoveL 294 to (-5.57, -1302.9, 0) mm, rotated rx 0 ry 90 rz 0 deg; joints [18.102, -79.513, 145.755, -160.345, 67.484, 172.212]
  MoveL 295 to (-5.57, -1302.9, 100) mm, rotated rx 0 ry 90 rz 0 deg; joints [18.102, -86.921, 143.552, -158.624, 58.479, 168.435]
  Set speed (1000.0 mm/s)
  MoveL 296 to (-5.57, -1274.17, 100) mm, rotated rx 0 ry 90 rz 0 deg; joints [16.471, -87.469, 144.139, -160.513, 58.203, 169.438]
  MoveL 297 to (-5.57, -1274.17, 0) mm, rotated rx 0 ry 90 rz 0 deg; joints [16.471, -79.973, 146.366, -162.117, 67.416, 172.936]
  MoveL 298 to (-5.57, -1274.17, 0) mm, rotated rx 0 ry 90 rz 0 deg; joints [16.471, -79.973, 146.366, -162.117, 67.416, 172.936]
  Set speed (50.0 mm/s)
  MoveL 299 to (43.17, -1325.29, 68.91) mm, rotated rx 0 ry 90 rz 0 deg; joints [18.447, -81.579, 140.581, -158.737, 60.755, 169.236]
  Set speed (1000.0 mm/s)
  MoveL 300 to (43.17, -1325.29, 68.91) mm, rotated rx 0 ry 90 rz 0 deg; joints [18.447, -81.579, 140.581, -158.737, 60.755, 169.236]
  MoveL 301 to (43.17, -1325.29, 168.91) mm, rotated rx 0 ry 90 rz 0 deg; joints [18.447, -87.683, 137.838, -156.518, 52.57, 165.209]
  Set speed (1000.0 mm/s)
  MoveL 302 to (38.44, -1305.95, 168.91) mm, rotated rx 0 ry 90 rz 0 deg; joints [17.492, -88.369, 138.556, -157.694, 52.361, 165.935]
  MoveL 303 to (38.44, -1305.95, 68.91) mm, rotated rx 0 ry 90 rz 0 deg; joints [17.492, -82.192, 141.328, -159.841, 60.707, 169.817]
  MoveL 304 to (38.44, -1305.95, 68.91) mm, rotated rx 0 ry 90 rz 0 deg; joints [17.492, -82.192, 141.328, -159.841, 60.707, 169.817]
  Set speed (50.0 mm/s)
  MoveL 305 to (-5.57, -1245.44, 0) mm, rotated rx 0 ry 90 rz 0 deg; joints [14.811, -80.394, 146.919, -163.918, 67.349, 173.665]
  Set speed (1000.0 mm/s)
  MoveL 306 to (-5.57, -1245.44, 0) mm, rotated rx 0 ry 90 rz 0 deg; joints [14.811, -80.394, 146.919, -163.918, 67.349, 173.665]
  MoveL 307 to (-5.57, -1245.44, 100) mm, rotated rx 0 ry 90 rz 0 deg; joints [14.811, -87.97, 144.671, -162.444, 57.942, 170.468]
  Set speed (1000.0 mm/s)
  MoveL 308 to (-5.57, -1216.71, 100) mm, rotated rx 0 ry 90 rz 0 deg; joints [13.126, -88.423, 145.144, -164.414, 57.699, 171.522]
  MoveL 309 to (-5.57, -1216.71, 0) mm, rotated rx 0 ry 90 rz 0 deg; joints [13.126, -80.773, 147.412, -165.747, 67.285, 174.398]
  MoveL 310 to (-5.57, -1216.71, 0) mm, rotated rx 0 ry 90 rz 0 deg; joints [13.126, -80.773, 147.412, -165.747, 67.285, 174.398]
  Set speed (50.0 mm/s)
  MoveL 311 to (33.7, -1286.62, 68.91) mm, rotated rx 0 ry 90 rz 0 deg; joints [16.517, -82.792, 142.051, -160.965, 60.655, 170.403]
  Set speed (1000.0 mm/s)
  MoveL 312 to (33.7, -1286.62, 68.91) mm, rotated rx 0 ry 90 rz 0 deg; joints [16.517, -82.792, 142.051, -160.965, 60.655, 170.403]
  MoveL 313 to (33.7, -1286.62, 168.91) mm, rotated rx 0 ry 90 rz 0 deg; joints [16.517, -89.042, 139.25, -158.897, 52.15, 166.677]
  Set speed (1000.0 mm/s)
  MoveL 314 to (28.97, -1267.28, 168.91) mm, rotated rx 0 ry 90 rz 0 deg; joints [15.522, -89.703, 139.919, -160.129, 51.936, 167.438]
  MoveL 315 to (28.97, -1267.28, 68.91) mm, rotated rx 0 ry 90 rz 0 deg; joints [15.522, -83.38, 142.75, -162.111, 60.599, 170.996]
  MoveL 316 to (28.97, -1267.28, 68.91) mm, rotated rx 0 ry 90 rz 0 deg; joints [15.522, -83.38, 142.75, -162.111, 60.599, 170.996]
  Set speed (50.0 mm/s)
  MoveL 317 to (-5.57, -1187.98, 0) mm, rotated rx 0 ry 90 rz 0 deg; joints [11.418, -81.108, 147.846, -167.602, 67.224, 175.136]
  Set speed (1000.0 mm/s)
  MoveL 318 to (-5.57, -1187.98, 0) mm, rotated rx 0 ry 90 rz 0 deg; joints [11.418, -81.108, 147.846, -167.602, 67.224, 175.136]
  MoveL 319 to (-5.57, -1187.98, 100) mm, rotated rx 0 ry 90 rz 0 deg; joints [11.418, -88.825, 145.56, -166.421, 57.476, 172.601]
  Set speed (1000.0 mm/s)
  MoveL 320 to (-5.57, -1159.25, 100) mm, rotated rx 0 ry 90 rz 0 deg; joints [9.689, -89.173, 145.918, -168.461, 57.279, 173.702]
  MoveL 321 to (-5.57, -1159.25, 0) mm, rotated rx 0 ry 90 rz 0 deg; joints [9.689, -81.399, 148.219, -169.479, 67.169, 175.878]
  MoveL 322 to (-5.57, -1159.25, 0) mm, rotated rx 0 ry 90 rz 0 deg; joints [9.689, -81.399, 148.219, -169.479, 67.169, 175.878]
  Set speed (50.0 mm/s)
  MoveL 323 to (24.24, -1247.95, 68.91) mm, rotated rx 0 ry 90 rz 0 deg; joints [14.508, -83.955, 143.425, -163.279, 60.541, 171.595]
  Set speed (1000.0 mm/s)
  MoveL 324 to (24.24, -1247.95, 68.91) mm, rotated rx 0 ry 90 rz 0 deg; joints [14.508, -83.955, 143.425, -163.279, 60.541, 171.595]
  MoveL 325 to (24.24, -1247.95, 168.91) mm, rotated rx 0 ry 90 rz 0 deg; joints [14.508, -90.349, 140.565, -161.39, 51.722, 168.217]
  Set speed (1000.0 mm/s)
  MoveL 326 to (19.51, -1228.61, 168.91) mm, rotated rx 0 ry 90 rz 0 deg; joints [13.474, -90.979, 141.186, -162.681, 51.508, 169.016]
  MoveL 327 to (19.51, -1228.61, 68.91) mm, rotated rx 0 ry 90 rz 0 deg; joints [13.474, -84.517, 144.075, -164.469, 60.48, 172.203]
  MoveL 328 to (19.51, -1228.61, 68.91) mm, rotated rx 0 ry 90 rz 0 deg; joints [13.474, -84.517, 144.075, -164.469, 60.48, 172.203]
  Set speed (50.0 mm/s)
  MoveL 329 to (-5.57, -1130.52, 0) mm, rotated rx 0 ry 90 rz 0 deg; joints [7.941, -81.643, 148.53, -171.376, 67.122, 176.625]
  Set speed (1000.0 mm/s)
  MoveL 330 to (-5.57, -1130.52, 0) mm, rotated rx 0 ry 90 rz 0 deg; joints [7.941, -81.643, 148.53, -171.376, 67.122, 176.625]
  MoveL 331 to (-5.57, -1130.52, 100) mm, rotated rx 0 ry 90 rz 0 deg; joints [7.941, -89.466, 146.216, -170.53, 57.109, 174.824]
  Set speed (1000.0 mm/s)
  MoveL 332 to (105.47, -1453.49, 168.91) mm, rotated rx 0 ry 90 rz 0 deg; joints [23.642, -81.146, 130.458, -150.001, 53.329, 160.976]
  MoveL 333 to (105.47, -1453.49, 68.91) mm, rotated rx 0 ry 90 rz 0 deg; joints [23.642, -75.717, 132.956, -152.5, 60.283, 165.53]
  MoveL 334 to (105.47, -1453.49, 68.91) mm, rotated rx 0 ry 90 rz 0 deg; joints [23.642, -75.717, 132.956, -152.5, 60.283, 165.53]
  Set speed (50.0 mm/s)
  MoveL 335 to (43.97, -1202.13, 68.91) mm, rotated rx 0 ry 90 rz 0 deg; joints [11.653, -83.424, 142.801, -166.522, 60.074, 173.182]
  Set speed (1000.0 mm/s)
  MoveL 336 to (43.97, -1202.13, 68.91) mm, rotated rx 0 ry 90 rz 0 deg; joints [11.653, -83.424, 142.801, -166.522, 60.074, 173.182]
  MoveL 337 to (43.97, -1202.13, 168.91) mm, rotated rx 0 ry 90 rz 0 deg; joints [11.653, -89.752, 139.969, -164.977, 51.194, 170.453]
  Set speed (1000.0 mm/s)
  MoveL 338 to (134.66, -1446.35, 168.91) mm, rotated rx 0 ry 90 rz 0 deg; joints [22.732, -79.702, 128.698, -150.962, 52.76, 161.429]
  MoveL 339 to (134.66, -1446.35, 68.91) mm, rotated rx 0 ry 90 rz 0 deg; joints [22.732, -74.414, 131.151, -153.386, 59.61, 165.776]
  MoveL 340 to (134.66, -1446.35, 68.91) mm, rotated rx 0 ry 90 rz 0 deg; joints [22.732, -74.414, 131.151, -153.386, 59.61, 165.776]
  Set speed (50.0 mm/s)
  MoveL 341 to (73.15, -1194.99, 68.91) mm, rotated rx 0 ry 90 rz 0 deg; joints [10.927, -81.815, 140.87, -167.314, 59.675, 173.516]
  Set speed (1000.0 mm/s)
  MoveL 342 to (73.15, -1194.99, 68.91) mm, rotated rx 0 ry 90 rz 0 deg; joints [10.927, -81.815, 140.87, -167.314, 59.675, 173.516]
  MoveL 343 to (73.15, -1194.99, 168.91) mm, rotated rx 0 ry 90 rz 0 deg; joints [10.927, -87.947, 138.116, -165.888, 51.03, 171.015]
  Set speed (1000.0 mm/s)
  MoveL 344 to (163.85, -1439.21, 168.91) mm, rotated rx 0 ry 90 rz 0 deg; joints [21.86, -78.26, 126.894, -151.873, 52.169, 161.848]
  MoveL 345 to (163.85, -1439.21, 68.91) mm, rotated rx 0 ry 90 rz 0 deg; joints [21.86, -73.108, 129.304, -154.228, 58.912, 166.001]
  MoveL 346 to (163.85, -1439.21, 68.91) mm, rotated rx 0 ry 90 rz 0 deg; joints [21.86, -73.108, 129.304, -154.228, 58.912, 166.001]
  Set speed (50.0 mm/s)
  MoveL 347 to (102.34, -1187.85, 68.91) mm, rotated rx 0 ry 90 rz 0 deg; joints [10.239, -80.232, 138.904, -168.06, 59.225, 173.825]
  Set speed (1000.0 mm/s)
  MoveL 348 to (102.34, -1187.85, 68.91) mm, rotated rx 0 ry 90 rz 0 deg; joints [10.239, -80.232, 138.904, -168.06, 59.225, 173.825]
  MoveL 349 to (102.34, -1187.85, 168.91) mm, rotated rx 0 ry 90 rz 0 deg; joints [10.239, -86.175, 136.223, -166.741, 50.808, 171.531]
  Set speed (1000.0 mm/s)
  MoveL 350 to (193.03, -1432.07, 168.91) mm, rotated rx 0 ry 90 rz 0 deg; joints [21.023, -76.817, 125.046, -152.737, 51.552, 162.233]
  MoveL 351 to (193.03, -1432.07, 68.91) mm, rotated rx 0 ry 90 rz 0 deg; joints [21.023, -71.799, 127.416, -155.029, 58.188, 166.208]
  MoveL 352 to (193.03, -1432.07, 68.91) mm, rotated rx 0 ry 90 rz 0 deg; joints [21.023, -71.799, 127.416, -155.029, 58.188, 166.208]
  Set speed (50.0 mm/s)
  MoveL 353 to (131.53, -1180.71, 68.91) mm, rotated rx 0 ry 90 rz 0 deg; joints [9.586, -78.673, 136.905, -168.765, 58.727, 174.112]
  Set speed (1000.0 mm/s)
  MoveL 354 to (131.53, -1180.71, 68.91) mm, rotated rx 0 ry 90 rz 0 deg; joints [9.586, -78.673, 136.905, -168.765, 58.727, 174.112]
  MoveL 355 to (131.53, -1180.71, 168.91) mm, rotated rx 0 ry 90 rz 0 deg; joints [9.586, -84.433, 134.291, -167.542, 50.529, 172.006]
  Set speed (1000.0 mm/s)
  MoveL 356 to (222.22, -1424.93, 168.91) mm, rotated rx 0 ry 90 rz 0 deg; joints [20.221, -75.374, 123.154, -153.556, 50.908, 162.587]
  MoveL 357 to (222.22, -1424.93, 68.91) mm, rotated rx 0 ry 90 rz 0 deg; joints [20.221, -70.485, 125.486, -155.789, 57.438, 166.396]
  MoveL 358 to (222.22, -1424.93, 68.91) mm, rotated rx 0 ry 90 rz 0 deg; joints [20.221, -70.485, 125.486, -155.789, 57.438, 166.396]
  Set speed (50.0 mm/s)
  MoveL 359 to (160.71, -1173.57, 68.91) mm, rotated rx 0 ry 90 rz 0 deg; joints [8.966, -77.132, 134.873, -169.432, 58.181, 174.382]
  Set speed (1000.0 mm/s)
  MoveL 360 to (160.71, -1173.57, 68.91) mm, rotated rx 0 ry 90 rz 0 deg; joints [8.966, -77.132, 134.873, -169.432, 58.181, 174.382]
  MoveL 361 to (160.71, -1173.57, 168.91) mm, rotated rx 0 ry 90 rz 0 deg; joints [8.966, -82.718, 132.321, -168.296, 50.196, 172.445]
  Set speed (1000.0 mm/s)
  MoveL 362 to (251.41, -1417.78, 168.91) mm, rotated rx 0 ry 90 rz 0 deg; joints [19.45, -73.928, 121.216, -154.331, 50.237, 162.913]
  MoveL 363 to (251.41, -1417.78, 68.91) mm, rotated rx 0 ry 90 rz 0 deg; joints [19.45, -69.166, 123.515, -156.511, 56.661, 166.567]
  MoveL 364 to (251.41, -1417.78, 68.91) mm, rotated rx 0 ry 90 rz 0 deg; joints [19.45, -69.166, 123.515, -156.511, 56.661, 166.567]
  Set speed (50.0 mm/s)
  MoveL 365 to (189.9, -1166.42, 68.91) mm, rotated rx 0 ry 90 rz 0 deg; joints [8.376, -75.608, 132.806, -170.064, 57.591, 174.637]
  Set speed (1000.0 mm/s)
  MoveL 366 to (189.9, -1166.42, 68.91) mm, rotated rx 0 ry 90 rz 0 deg; joints [8.376, -75.608, 132.806, -170.064, 57.591, 174.637]
  MoveL 367 to (189.9, -1166.42, 168.91) mm, rotated rx 0 ry 90 rz 0 deg; joints [8.376, -81.025, 130.312, -169.007, 49.811, 172.855]
  Set speed (1000.0 mm/s)
  MoveL 368 to (280.59, -1410.64, 168.91) mm, rotated rx 0 ry 90 rz 0 deg; joints [18.709, -72.48, 119.233, -155.064, 49.538, 163.21]
  MoveL 369 to (280.59, -1410.64, 68.91) mm, rotated rx 0 ry 90 rz 0 deg; joints [18.709, -67.841, 121.5, -157.196, 55.856, 166.722]
  MoveL 370 to (280.59, -1410.64, 68.91) mm, rotated rx 0 ry 90 rz 0 deg; joints [18.709, -67.841, 121.5, -157.196, 55.856, 166.722]
  Set speed (50.0 mm/s)
  MoveL 371 to (219.09, -1159.28, 68.91) mm, rotated rx 0 ry 90 rz 0 deg; joints [7.815, -74.097, 130.706, -170.665, 56.959, 174.878]
  Set speed (1000.0 mm/s)
  MoveL 372 to (219.09, -1159.28, 68.91) mm, rotated rx 0 ry 90 rz 0 deg; joints [7.815, -74.097, 130.706, -170.665, 56.959, 174.878]
  MoveL 373 to (219.09, -1159.28, 168.91) mm, rotated rx 0 ry 90 rz 0 deg; joints [7.815, -79.352, 128.264, -169.68, 49.375, 173.238]
  Set speed (1000.0 mm/s)
  MoveL 374 to (309.78, -1403.5, 168.91) mm, rotated rx 0 ry 90 rz 0 deg; joints [17.998, -71.027, 117.202, -155.758, 48.809, 163.482]
  MoveL 375 to (309.78, -1403.5, 68.91) mm, rotated rx 0 ry 90 rz 0 deg; joints [17.998, -66.507, 119.442, -157.846, 55.024, 166.863]
  MoveL 376 to (309.78, -1403.5, 68.91) mm, rotated rx 0 ry 90 rz 0 deg; joints [17.998, -66.507, 119.442, -157.846, 55.024, 166.863]
  Set speed (50.0 mm/s)
  MoveL 377 to (248.28, -1152.14, 68.91) mm, rotated rx 0 ry 90 rz 0 deg; joints [7.28, -72.596, 128.57, -171.237, 56.285, 175.11]
  Set speed (1000.0 mm/s)
  MoveL 378 to (248.28, -1152.14, 68.91) mm, rotated rx 0 ry 90 rz 0 deg; joints [7.28, -72.596, 128.57, -171.237, 56.285, 175.11]
  MoveL 379 to (248.28, -1152.14, 168.91) mm, rotated rx 0 ry 90 rz 0 deg; joints [7.28, -77.695, 126.177, -170.317, 48.889, 173.599]
  Set speed (1000.0 mm/s)
  MoveL 380 to (338.97, -1396.36, 168.91) mm, rotated rx 0 ry 90 rz 0 deg; joints [17.314, -69.568, 115.124, -156.412, 48.05, 163.728]
  MoveL 381 to (338.97, -1396.36, 68.91) mm, rotated rx 0 ry 90 rz 0 deg; joints [17.314, -65.165, 117.338, -158.463, 54.163, 166.989]
  MoveL 382 to (338.97, -1396.36, 68.91) mm, rotated rx 0 ry 90 rz 0 deg; joints [17.314, -65.165, 117.338, -158.463, 54.163, 166.989]
  Set speed (50.0 mm/s)
  MoveL 383 to (277.46, -1145, 68.91) mm, rotated rx 0 ry 90 rz 0 deg; joints [6.77, -71.103, 126.399, -171.783, 55.572, 175.333]
  Set speed (1000.0 mm/s)
  MoveL 384 to (277.46, -1145, 68.91) mm, rotated rx 0 ry 90 rz 0 deg; joints [6.77, -71.103, 126.399, -171.783, 55.572, 175.333]
  MoveL 385 to (277.46, -1145, 168.91) mm, rotated rx 0 ry 90 rz 0 deg; joints [6.77, -76.052, 124.049, -170.924, 48.355, 173.94]
  Set speed (1000.0 mm/s)
  MoveL 386 to (368.16, -1389.22, 168.91) mm, rotated rx 0 ry 90 rz 0 deg; joints [16.656, -68.101, 112.996, -157.029, 47.259, 163.951]
  MoveL 387 to (368.16, -1389.22, 68.91) mm, rotated rx 0 ry 90 rz 0 deg; joints [16.656, -63.812, 115.188, -159.046, 53.272, 167.101]
  MoveL 388 to (368.16, -1389.22, 68.91) mm, rotated rx 0 ry 90 rz 0 deg; joints [16.656, -63.812, 115.188, -159.046, 53.272, 167.101]
  Set speed (50.0 mm/s)
  MoveL 389 to (306.65, -1137.86, 68.91) mm, rotated rx 0 ry 90 rz 0 deg; joints [6.283, -69.615, 124.19, -172.305, 54.819, 175.548]
  Set speed (1000.0 mm/s)
  MoveL 390 to (306.65, -1137.86, 68.91) mm, rotated rx 0 ry 90 rz 0 deg; joints [6.283, -69.615, 124.19, -172.305, 54.819, 175.548]
  MoveL 391 to (306.65, -1137.86, 168.91) mm, rotated rx 0 ry 90 rz 0 deg; joints [6.283, -74.42, 121.88, -171.501, 47.775, 174.265]
  Set speed (1000.0 mm/s)
  MoveL 392 to (397.34, -1382.08, 168.91) mm, rotated rx 0 ry 90 rz 0 deg; joints [16.023, -66.626, 110.817, -157.609, 46.436, 164.149]
  MoveL 393 to (397.34, -1382.08, 68.91) mm, rotated rx 0 ry 90 rz 0 deg; joints [16.023, -62.447, 112.99, -159.597, 52.351, 167.2]
  MoveL 394 to (397.34, -1382.08, 68.91) mm, rotated rx 0 ry 90 rz 0 deg; joints [16.023, -62.447, 112.99, -159.597, 52.351, 167.2]
  Set speed (50.0 mm/s)
  MoveL 395 to (335.84, -1130.72, 68.91) mm, rotated rx 0 ry 90 rz 0 deg; joints [5.818, -68.13, 121.942, -172.805, 54.028, 175.759]
  Set speed (1000.0 mm/s)
  MoveL 396 to (335.84, -1130.72, 68.91) mm, rotated rx 0 ry 90 rz 0 deg; joints [5.818, -68.13, 121.942, -172.805, 54.028, 175.759]
  MoveL 397 to (335.84, -1130.72, 168.91) mm, rotated rx 0 ry 90 rz 0 deg; joints [5.818, -72.795, 119.668, -172.052, 47.149, 174.576]
  Set speed (1000.0 mm/s)
  MoveL 398 to (426.53, -1374.93, 168.91) mm, rotated rx 0 ry 90 rz 0 deg; joints [15.413, -65.139, 108.584, -158.153, 45.579, 164.325]
  MoveL 399 to (426.53, -1374.93, 68.91) mm, rotated rx 0 ry 90 rz 0 deg; joints [15.413, -61.068, 110.741, -160.118, 51.4, 167.286]
  MoveL 400 to (426.53, -1374.93, 68.91) mm, rotated rx 0 ry 90 rz 0 deg; joints [15.413, -61.068, 110.741, -160.118, 51.4, 167.286]
  Set speed (50.0 mm/s)
  MoveL 401 to (365.02, -1123.57, 68.91) mm, rotated rx 0 ry 90 rz 0 deg; joints [5.373, -66.644, 119.654, -173.284, 53.2, 175.965]
  Set speed (1000.0 mm/s)
  MoveL 402 to (365.02, -1123.57, 68.91) mm, rotated rx 0 ry 90 rz 0 deg; joints [5.373, -66.644, 119.654, -173.284, 53.2, 175.965]
  MoveL 403 to (365.02, -1123.57, 168.91) mm, rotated rx 0 ry 90 rz 0 deg; joints [5.373, -71.176, 117.413, -172.58, 46.477, 174.875]
